(* IEC 61131-3 sources: RL_MAR/experiments/comparison/llm4plc/results/gpt-4o-mini_20260506_100619/20260506_102052, 3 files *)

(* ---- generated_code_iteration_0.st ---- *)
ructured-text
START_ST
FUNCTION_BLOCK FishTankControl
VAR_INPUT
    OxygenLevel : REAL; (* Input for oxygen level in the tank *)
    WaterTemperature : REAL; (* Input for water temperature *)
    FeedingTime : TIME; (* Time for scheduled feeding *)
    CurrentTime : TIME; (* Current system time *)
END_VAR
VAR_OUTPUT
    OxygenValve : BOOL; (* Output to control oxygen supply *)
    Heater : BOOL; (* Output to control the heater *)
    Feeder : BOOL; (* Output to control the fish feeder *)
END_VAR
VAR
    state : INT; (* Current state variable *)
    prevState : INT; (* Previous state variable *)
END_VAR

(* State definitions *)
STATE_MONITORING : INT := 0;
STATE_OPEN_OXYGEN_VALVE : INT := 1;
STATE_TURN_ON_HEATER : INT := 2;
STATE_OPERATE_FEEDER : INT := 3;

(* Initialize outputs *)
OxygenValve := FALSE;
Heater := FALSE;
Feeder := FALSE;

(* State machine logic *)
CASE state OF
    STATE_MONITORING:
        (* Check conditions for state transitions *)
        IF OxygenLevel < 5.0 THEN
            state := STATE_OPEN_OXYGEN_VALVE;
        ELSIF WaterTemperature < 25.0 THEN
            state := STATE_TURN_ON_HEATER;
        ELSIF CurrentTime >= FeedingTime THEN
            state := STATE_OPERATE_FEEDER;
        END_IF;

        (* Set outputs for monitoring state *)
        OxygenValve := FALSE;
        Heater := FALSE;
        Feeder := FALSE;

    STATE_OPEN_OXYGEN_VALVE:
        (* Check condition to return to monitoring state *)
        IF OxygenLevel >= 5.0 THEN
            state := STATE_MONITORING;
        END_IF;

        (* Set outputs for opening oxygen valve state *)
        OxygenValve := TRUE;
        Heater := FALSE;
        Feeder := FALSE;

    STATE_TURN_ON_HEATER:
        (* Check condition to return to monitoring state *)
        IF WaterTemperature >= 25.0 THEN
            state := STATE_MONITORING;
        END_IF;

        (* Set outputs for turning on heater state *)
        OxygenValve := FALSE;
        Heater := TRUE;
        Feeder := FALSE;

    STATE_OPERATE_FEEDER:
        (* Check condition to return to monitoring state *)
        IF CurrentTime < FeedingTime THEN
            state := STATE_MONITORING;
        END_IF;

        (* Set outputs for operating feeder state *)
        OxygenValve := FALSE;
        Heater := FALSE;
        Feeder := TRUE;

    ELSE
        (* Default case to ensure valid state *)
        state := STATE_MONITORING;
END_CASE;

END_FUNCTION_BLOCK
END_ST

(* ---- generated_code_iteration_1.st ---- *)
START_REASON
The errors in the original Structured Text (ST) code occurred due to the incorrect use of variable section terminators. Specifically, the variable section was incorrectly closed with "END_VAR_OUTPUT" and "END_VAR_INPUT", which are not valid in ST. The correct terminator is "END_VAR". Additionally, the state definitions should be declared within the variable section to ensure proper scope and initialization. The overall structure of the function block must be maintained while correcting these issues.
END_REASON

START_ST
FUNCTION_BLOCK FishTankControl
VAR_INPUT
    OxygenLevel : REAL; (* Input for oxygen level in the tank *)
    WaterTemperature : REAL; (* Input for water temperature *)
    FeedingTime : TIME; (* Time for scheduled feeding *)
    CurrentTime : TIME; (* Current system time *)
END_VAR
VAR_OUTPUT
    OxygenValve : BOOL; (* Output to control oxygen supply *)
    Heater : BOOL; (* Output to control the heater *)
    Feeder : BOOL; (* Output to control the fish feeder *)
END_VAR
VAR
    state : INT; (* Current state variable *)
    prevState : INT; (* Previous state variable *)
    STATE_MONITORING : INT := 0; (* State definitions *)
    STATE_OPEN_OXYGEN_VALVE : INT := 1;
    STATE_TURN_ON_HEATER : INT := 2;
    STATE_OPERATE_FEEDER : INT := 3;
END_VAR

(* Initialize outputs *)
OxygenValve := FALSE;
Heater := FALSE;
Feeder := FALSE;

(* State machine logic *)
CASE state OF
    STATE_MONITORING:
        (* Check conditions for state transitions *)
        IF OxygenLevel < 5.0 THEN
            state := STATE_OPEN_OXYGEN_VALVE;
        ELSIF WaterTemperature < 25.0 THEN
            state := STATE_TURN_ON_HEATER;
        ELSIF CurrentTime >= FeedingTime THEN
            state := STATE_OPERATE_FEEDER;
        END_IF;

        (* Set outputs for monitoring state *)
        OxygenValve := FALSE;
        Heater := FALSE;
        Feeder := FALSE;

    STATE_OPEN_OXYGEN_VALVE:
        (* Check condition to return to monitoring state *)
        IF OxygenLevel >= 5.0 THEN
            state := STATE_MONITORING;
        END_IF;

        (* Set outputs for opening oxygen valve state *)
        OxygenValve := TRUE;
        Heater := FALSE;
        Feeder := FALSE;

    STATE_TURN_ON_HEATER:
        (* Check condition to return to monitoring state *)
        IF WaterTemperature >= 25.0 THEN
            state := STATE_MONITORING;
        END_IF;

        (* Set outputs for turning on heater state *)
        OxygenValve := FALSE;
        Heater := TRUE;
        Feeder := FALSE;

    STATE_OPERATE_FEEDER:
        (* Check condition to return to monitoring state *)
        IF CurrentTime < FeedingTime THEN
            state := STATE_MONITORING;
        END_IF;

        (* Set outputs for operating feeder state *)
        OxygenValve := FALSE;
        Heater := FALSE;
        Feeder := TRUE;

    ELSE
        (* Default case to ensure valid state *)
        state := STATE_MONITORING;
END_CASE;

END_FUNCTION_BLOCK
END_ST

(* ---- generated_code_iteration_2.st ---- *)
START_REASON
The errors in the original Structured Text (ST) code occurred due to the incorrect use of variable section terminators. Specifically, the variable section was incorrectly closed with "END_VAR_OUTPUT" and "END_VAR_INPUT", which are not valid in ST. The correct terminator is "END_VAR". Additionally, the state definitions should be declared within the variable section to ensure proper scope and initialization. The overall structure of the function block must be maintained while correcting these issues. Furthermore, the CODESYS compiler validation error indicates that the CASE statement requires constant integer values for its labels, which were not properly defined in the original code. This necessitates ensuring that the state variables used in the CASE statement are correctly defined and utilized.
END_REASON

START_ST
FUNCTION_BLOCK FishTankControl
VAR_INPUT
    OxygenLevel : REAL; (* Input for oxygen level in the tank *)
    WaterTemperature : REAL; (* Input for water temperature *)
    FeedingTime : TIME; (* Time for scheduled feeding *)
    CurrentTime : TIME; (* Current system time *)
END_VAR
VAR_OUTPUT
    OxygenValve : BOOL; (* Output to control oxygen supply *)
    Heater : BOOL; (* Output to control the heater *)
    Feeder : BOOL; (* Output to control the fish feeder *)
END_VAR
VAR
    state : INT; (* Current state variable *)
    prevState : INT; (* Previous state variable *)
    STATE_MONITORING : INT := 0; (* State definitions *)
    STATE_OPEN_OXYGEN_VALVE : INT := 1;
    STATE_TURN_ON_HEATER : INT := 2;
    STATE_OPERATE_FEEDER : INT := 3;
END_VAR

(* Initialize outputs *)
OxygenValve := FALSE;
Heater := FALSE;
Feeder := FALSE;

(* State machine logic *)
CASE state OF
    0: (* STATE_MONITORING *)
        (* Check conditions for state transitions *)
        IF OxygenLevel < 5.0 THEN
            state := STATE_OPEN_OXYGEN_VALVE;
        ELSIF WaterTemperature < 25.0 THEN
            state := STATE_TURN_ON_HEATER;
        ELSIF CurrentTime >= FeedingTime THEN
            state := STATE_OPERATE_FEEDER;
        END_IF;

        (* Set outputs for monitoring state *)
        OxygenValve := FALSE;
        Heater := FALSE;
        Feeder := FALSE;

    1: (* STATE_OPEN_OXYGEN_VALVE *)
        (* Check condition to return to monitoring state *)
        IF OxygenLevel >= 5.0 THEN
            state := STATE_MONITORING;
        END_IF;

        (* Set outputs for opening oxygen valve state *)
        OxygenValve := TRUE;
        Heater := FALSE;
        Feeder := FALSE;

    2: (* STATE_TURN_ON_HEATER *)
        (* Check condition to return to monitoring state *)
        IF WaterTemperature >= 25.0 THEN
            state := STATE_MONITORING;
        END_IF;

        (* Set outputs for turning on heater state *)
        OxygenValve := FALSE;
        Heater := TRUE;
        Feeder := FALSE;

    3: (* STATE_OPERATE_FEEDER *)
        (* Check condition to return to monitoring state *)
        IF CurrentTime < FeedingTime THEN
            state := STATE_MONITORING;
        END_IF;

        (* Set outputs for operating feeder state *)
        OxygenValve := FALSE;
        Heater := FALSE;
        Feeder := TRUE;

    ELSE
        (* Default case to ensure valid state *)
        state := STATE_MONITORING;
END_CASE;

END_FUNCTION_BLOCK
END_ST
